Fanuc KAREL source: inv_nolg.kl

PROGRAM INV_NOLG
%INVISIBLE
%NOLOCKGROUP
VAR
	I : INTEGER
BEGIN
	I = 1
	WRITE('I = ', I, CR)
END INV_NOLG
